# EPICS autosave request: iocBoot/gmca_23o_ioc1/dbSave/digital_IO_24_bo.req
%
% This request file stores settings for PMAC digital out
%

$(P)0.VAL
$(P)1.VAL
$(P)2.VAL
$(P)3.VAL
$(P)4.VAL
$(P)5.VAL
$(P)6.VAL
$(P)7.VAL
$(P)8.VAL
$(P)9.VAL
$(P)10.VAL
$(P)11.VAL
$(P)12.VAL
$(P)13.VAL
$(P)14.VAL
$(P)15.VAL
$(P)16.VAL
$(P)17.VAL
$(P)18.VAL
$(P)19.VAL
$(P)20.VAL
$(P)21.VAL
$(P)22.VAL
$(P)23.VAL
